FUNCTION alg_a_x2distributing : BOOL
VAR_INPUT
	state: STATE;
END_VAR

alg_a_x2distributing := state.dvar_M_example_controller_a_x2distributing;

END_FUNCTION

(* stored: Version 1.1.0.1, ProductVersion 3.1.4022.18
   POU alg_a_x2distributing: Id {49790717-d0e2-4214-a3f4-4ed080de9561}, SpecialFunc None *)
